DATA_BLOCK "FB_StartPrecheck_DB"
{ S7_Optimized_Access := 'TRUE' }
VERSION : 0.4
NON_RETAIN
"FB_StartPrecheck"

BEGIN

END_DATA_BLOCK

